VAR_GLOBAL
END_VAR


VAR_GLOBAL CONSTANT
	maxNumTasks: UINT := 20; //max number of tasks in the station.
END_VAR

(* stored: Version 1.1.0.1, ProductVersion 3.1.4024.12
   GVL Tasks: Id {d10f62d0-f326-46f1-900e-be5b5304ea05} *)
